RoboDK station: M301_01.rdk

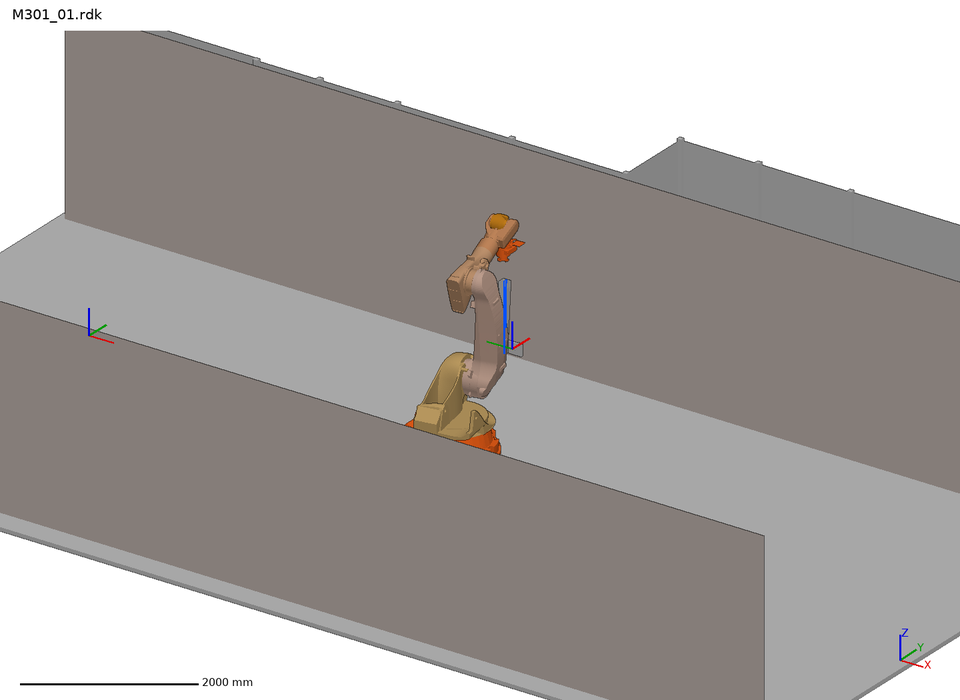
[picture v0: the station drawn from its stored meshes, robots at their saved joint values, targets as dots, program paths as lines]
Station CTTLab. Poses are relative to the parent item; angles as X-Y-Z fixed-axis rotations.
  - object PLANCHER at (0, 0, 0) mm, size 14365 x 8134 x 50 mm, geometry from PLANCHER.STL
  - object BARRIERE_POTEAU at (0, 0, 0) mm, size 13974 x 1274 x 2640 mm, geometry from BARRIERE_POTEAU.STL
  - object BARRIERE_GRILLAGE at (0, 0, 0) mm, size 13811.6 x 1129 x 2475 mm, geometry from BARRIERE_GRILLAGE.STL
  - object BARRIERE_IMMATERIELLE at (0, 0, 0) mm, size 14165 x 6570 x 2640 mm, geometry from BARRIERE_IMMATERIELLE.STL
  - frame World Base at (0, 0, 2.5) mm
    - robot Linear Rail: 1 axes
        modified DH rows (alpha deg, a mm, theta deg, d mm): 0, 0, 0, 0 linear
        base shift (0, 0, 0) mm, rotated rx 0 ry 90 rz 0 deg
        joint limits [0] to [7000]; home [0]; saved at [5000]
      - robot KUKA KR 100 HA: 6 axes
          modified DH rows (alpha deg, a mm, theta deg, d mm): 0, 0, 0, 750; -90, 350, 0, 0; 0, 1250, -90, 0; -90, -45, 0, 1000; 90, 0, 0, 0; -90, 0, 180, 210
          joint limits [-185, -120, -119, -350, -125, -350] to [185, 70, 155, 350, 125, 350]; home [0, -90, 90, 0, 0, 0]; saved at [-97.744, -95.279, 76.837, 0, 108.443, -187.744]
        - tool Tool 1, TCP at (13, 8, 496) mm, size 290.8 x 416.4 x 279.8 mm, geometry from OUTIL.STL
          - object M301_01 at (0, 0, 0) mm, size 101.6 x 101.6 x 914.4 mm, geometry from M301_01.stl
  - frame Camera base at (4846.59, 1350.74, 651.46) mm, rotated rx 0 ry 0 rz 90 deg
    - object Camera at (0, 0, 0) mm, rotated rx 90 ry 0 rz 90 deg, size 220 x 170 x 50 mm, geometry from Camera.stl
    - target Approach target (Cartesian target) at (-112.7, 0, 313.4) mm, rotated rx -180 ry 0 rz -90 deg; joints [-97.607, -91.723, 108.46, 0, 73.263, 82.393, 5000] of KUKA KR 100 HA
    - target Target 0 (Cartesian target) at (-112.7, 0, 881.94) mm, rotated rx -180 ry 0 rz -90 deg; joints [-97.607, -92.983, 76.617, 0, 106.366, 82.393, 5000] of KUKA KR 100 HA
    - target Target 1 (Cartesian target) at (-124.95, 0, 850.56) mm, rotated rx -180 ry 0 rz -90 deg; joints [-97.744, -94.315, 79.678, 0.115, 103.822, 82.256, 5000] of KUKA KR 100 HA
    - target Target 2 (Cartesian target) at (-139.47, 0, 817.45) mm, rotated rx -177.14 ry 0 rz -90 deg; joints [-97.914, -95.806, 82.96, 0.254, 101.05, 82.172, 5000] of KUKA KR 100 HA
    - target Target 3 (Cartesian target) at (-154.54, 0, 817.31) mm, rotated rx -177.14 ry 0 rz -90 deg; joints [-98.102, -97.065, 84.055, 0.41, 100.176, 81.98, 5000] of KUKA KR 100 HA
    - target Target 4 (Cartesian target) at (-154.54, 0, 785.81) mm, rotated rx -177.14 ry 0 rz -90 deg; joints [-98.102, -97.304, 86.085, 0.408, 98.386, 81.967, 5000] of KUKA KR 100 HA
    - target Target 5 (Cartesian target) at (-154.54, 0, 785.81) mm, rotated rx -177.14 ry 0 rz -90 deg; joints [-98.102, -97.304, 86.085, 0.408, 98.386, 81.967, 5000] of KUKA KR 100 HA
    - target Target 6 (Cartesian target) at (-154.54, 0, 754.31) mm, rotated rx -177.14 ry 0 rz -90 deg; joints [-98.102, -97.499, 88.067, 0.406, 96.598, 81.955, 5000] of KUKA KR 100 HA
    - target Target 7 (Cartesian target) at (-154.54, 0, 754.31) mm, rotated rx -177.14 ry 0 rz -90 deg; joints [-98.102, -97.499, 88.067, 0.406, 96.598, 81.955, 5000] of KUKA KR 100 HA
    - target Target 8 (Cartesian target) at (-154.54, 0, 722.81) mm, rotated rx -177.14 ry 0 rz -90 deg; joints [-98.102, -97.649, 90.006, 0.405, 94.81, 81.942, 5000] of KUKA KR 100 HA
    - target Target 9 (Cartesian target) at (-154.54, 0, 722.81) mm, rotated rx -177.14 ry 0 rz -90 deg; joints [-98.102, -97.649, 90.006, 0.405, 94.81, 81.942, 5000] of KUKA KR 100 HA
    - target Target 10 (Cartesian target) at (-154.54, 0, 691.3) mm, rotated rx -177.14 ry 0 rz -90 deg; joints [-98.102, -97.754, 91.901, 0.404, 93.019, 81.929, 5000] of KUKA KR 100 HA
    - target Target 11 (Cartesian target) at (-154.54, 0, 691.3) mm, rotated rx -177.14 ry 0 rz -90 deg; joints [-98.102, -97.754, 91.901, 0.404, 93.019, 81.929, 5000] of KUKA KR 100 HA
    - target Target 12 (Cartesian target) at (-154.54, 0, 659.8) mm, rotated rx -177.14 ry 0 rz -90 deg; joints [-98.102, -97.815, 93.756, 0.403, 91.225, 81.917, 5000] of KUKA KR 100 HA
    - target Target 13 (Cartesian target) at (-154.54, 0, 659.8) mm, rotated rx -177.14 ry 0 rz -90 deg; joints [-98.102, -97.815, 93.756, 0.403, 91.225, 81.917, 5000] of KUKA KR 100 HA
    - target Target 14 (Cartesian target) at (-154.54, 0, 628.3) mm, rotated rx -177.14 ry 0 rz -90 deg; joints [-98.102, -97.829, 95.571, 0.403, 89.424, 81.904, 5000] of KUKA KR 100 HA
    - target Target 15 (Cartesian target) at (-154.54, 0, 628.3) mm, rotated rx -177.14 ry 0 rz -90 deg; joints [-98.102, -97.829, 95.571, 0.403, 89.424, 81.904, 5000] of KUKA KR 100 HA
    - target Target 16 (Cartesian target) at (-154.54, 0, 596.8) mm, rotated rx -177.14 ry 0 rz -90 deg; joints [-98.102, -97.798, 97.349, 0.404, 87.615, 81.891, 5000] of KUKA KR 100 HA
    - target Target 17 (Cartesian target) at (-154.54, 0, 596.8) mm, rotated rx -177.14 ry 0 rz -90 deg; joints [-98.102, -97.798, 97.349, 0.404, 87.615, 81.891, 5000] of KUKA KR 100 HA
    - target Target 18 (Cartesian target) at (-154.54, 0, 565.3) mm, rotated rx -177.14 ry 0 rz -90 deg; joints [-98.102, -97.72, 99.09, 0.404, 85.797, 81.878, 5000] of KUKA KR 100 HA
    - target Target 19 (Cartesian target) at (-154.54, 0, 565.3) mm, rotated rx -177.14 ry 0 rz -90 deg; joints [-98.102, -97.72, 99.09, 0.404, 85.797, 81.878, 5000] of KUKA KR 100 HA
    - target Target 20 (Cartesian target) at (-154.54, 0, 533.8) mm, rotated rx -177.14 ry 0 rz -90 deg; joints [-98.102, -97.595, 100.795, 0.405, 83.966, 81.865, 5000] of KUKA KR 100 HA
    - target Target 21 (Cartesian target) at (-154.54, 0, 533.8) mm, rotated rx -177.14 ry 0 rz -90 deg; joints [-98.102, -97.595, 100.795, 0.405, 83.966, 81.865, 5000] of KUKA KR 100 HA
    - target Target 22 (Cartesian target) at (-154.54, 0, 502.3) mm, rotated rx -177.14 ry 0 rz -90 deg; joints [-98.102, -97.421, 102.465, 0.407, 82.122, 81.852, 5000] of KUKA KR 100 HA
    - target Target 23 (Cartesian target) at (-154.54, 0, 502.3) mm, rotated rx -177.14 ry 0 rz -90 deg; joints [-98.102, -97.421, 102.465, 0.407, 82.122, 81.852, 5000] of KUKA KR 100 HA
    - target Target 24 (Cartesian target) at (-154.54, 0, 470.79) mm, rotated rx -177.14 ry 0 rz -90 deg; joints [-98.102, -97.198, 104.102, 0.409, 80.263, 81.839, 5000] of KUKA KR 100 HA
    - target Target 25 (Cartesian target) at (-154.54, 0, 470.79) mm, rotated rx -177.14 ry 0 rz -90 deg; joints [-98.102, -97.198, 104.102, 0.409, 80.263, 81.839, 5000] of KUKA KR 100 HA
    - target Target 26 (Cartesian target) at (-154.54, 0, 439.29) mm, rotated rx -177.14 ry 0 rz -90 deg; joints [-98.102, -96.924, 105.704, 0.412, 78.387, 81.825, 5000] of KUKA KR 100 HA
    - target Target 27 (Cartesian target) at (-154.54, 0, 439.29) mm, rotated rx -177.14 ry 0 rz -90 deg; joints [-98.102, -96.924, 105.704, 0.412, 78.387, 81.825, 5000] of KUKA KR 100 HA
    - target Target 28 (Cartesian target) at (-154.54, 0, 407.79) mm, rotated rx -177.14 ry 0 rz -90 deg; joints [-98.102, -96.599, 107.273, 0.415, 76.492, 81.811, 5000] of KUKA KR 100 HA
    - target Target 29 (Cartesian target) at (-154.54, 0, 407.79) mm, rotated rx -177.14 ry 0 rz -90 deg; joints [-98.102, -96.599, 107.273, 0.415, 76.492, 81.811, 5000] of KUKA KR 100 HA
    - target Target 30 (Cartesian target) at (-154.54, 0, 376.29) mm, rotated rx -177.14 ry 0 rz -90 deg; joints [-98.102, -96.22, 108.809, 0.418, 74.578, 81.797, 5000] of KUKA KR 100 HA
    - target Target 31 (Cartesian target) at (-154.54, 0, 376.29) mm, rotated rx -177.14 ry 0 rz -90 deg; joints [-98.102, -96.22, 108.809, 0.418, 74.578, 81.797, 5000] of KUKA KR 100 HA
    - target Target 32 (Cartesian target) at (-154.54, 0, 344.79) mm, rotated rx -177.14 ry 0 rz -90 deg; joints [-98.102, -95.787, 110.312, 0.422, 72.642, 81.782, 5000] of KUKA KR 100 HA
    - target Target 33 (Cartesian target) at (-154.54, 0, 344.79) mm, rotated rx -177.14 ry 0 rz -90 deg; joints [-98.102, -95.787, 110.312, 0.422, 72.642, 81.782, 5000] of KUKA KR 100 HA
    - target Target 34 (Cartesian target) at (-154.54, 0, 313.29) mm, rotated rx -177.14 ry 0 rz -90 deg; joints [-98.102, -95.298, 111.781, 0.427, 70.683, 81.767, 5000] of KUKA KR 100 HA
    - target Target 35 (Cartesian target) at (-154.54, 0, 313.29) mm, rotated rx -177.14 ry 0 rz -90 deg; joints [-98.102, -95.298, 111.781, 0.427, 70.683, 81.767, 5000] of KUKA KR 100 HA
    - target Target 36 (Cartesian target) at (-154.54, 0, 281.79) mm, rotated rx -177.14 ry 0 rz -90 deg; joints [-98.102, -94.751, 113.218, 0.433, 68.7, 81.751, 5000] of KUKA KR 100 HA
    - target Target 37 (Cartesian target) at (-154.54, 0, 281.79) mm, rotated rx -177.14 ry 0 rz -90 deg; joints [-98.102, -94.751, 113.218, 0.433, 68.7, 81.751, 5000] of KUKA KR 100 HA
    - target Target 38 (Cartesian target) at (-154.54, 0, 250.29) mm, rotated rx -177.14 ry 0 rz -90 deg; joints [-98.102, -94.146, 114.621, 0.439, 66.691, 81.734, 5000] of KUKA KR 100 HA
    - target Target 39 (Cartesian target) at (-154.54, 0, 218.78) mm, rotated rx -177.14 ry 0 rz -90 deg; joints [-98.102, -93.479, 115.99, 0.446, 64.656, 81.717, 5000] of KUKA KR 100 HA
    - target Target 40 (Cartesian target) at (-154.54, 0, 218.78) mm, rotated rx -177.14 ry 0 rz -90 deg; joints [-98.102, -93.479, 115.99, 0.446, 64.656, 81.717, 5000] of KUKA KR 100 HA
    - target Target 41 (Cartesian target) at (-154.54, 0, 187.28) mm, rotated rx -177.14 ry 0 rz -90 deg; joints [-98.102, -92.751, 117.325, 0.454, 62.593, 81.699, 5000] of KUKA KR 100 HA
    - target Target 42 (Cartesian target) at (-154.54, 0, 187.28) mm, rotated rx -177.14 ry 0 rz -90 deg; joints [-98.102, -92.751, 117.325, 0.454, 62.593, 81.699, 5000] of KUKA KR 100 HA
    - target Target 43 (Cartesian target) at (-154.54, 0, 155.78) mm, rotated rx -177.14 ry 0 rz -90 deg; joints [81.898, -118.157, -84.385, 0.446, -64.624, -98.283, 5000] of KUKA KR 100 HA
    - target Target 44 (Cartesian target) at (-154.54, 0, 155.78) mm, rotated rx -177.14 ry 0 rz -90 deg; joints [81.898, -118.157, -84.385, 0.446, -64.624, -98.283, 5000] of KUKA KR 100 HA
    - target Target 45 (Cartesian target) at (-154.54, 0, 124.28) mm, rotated rx -177.14 ry 0 rz -90 deg; joints [81.898, -118.674, -85.469, 0.452, -63.024, -98.297, 5000] of KUKA KR 100 HA
    - target Target 46 (Cartesian target) at (-154.54, 0, 124.28) mm, rotated rx -177.14 ry 0 rz -90 deg; joints [81.898, -118.674, -85.469, 0.452, -63.024, -98.297, 5000] of KUKA KR 100 HA
    - target Target 47 (Cartesian target) at (-154.54, 0, 92.78) mm, rotated rx -177.14 ry 0 rz -90 deg; joints [81.898, -119.227, -86.504, 0.459, -61.436, -98.312, 5000] of KUKA KR 100 HA
    - target Target 48 (Cartesian target) at (-152.66, 0, 92.8) mm, rotated rx -177.14 ry 0 rz -90 deg; joints [82.007, -119.904, -85.364, 0.266, -63.062, -98.187, 5000] of KUKA KR 100 HA
    - target Target 49 (Cartesian target) at (-151.82, 0, 63.93) mm, rotated rx -180 ry 0 rz -90 deg; joints [-97.923, -88.095, 120.951, 0.152, 56.229, 82.077, 5000] of KUKA KR 100 HA
    - target Target 50 (Cartesian target) at (-150.8, 0, 32.46) mm, rotated rx -180 ry 0 rz -90 deg; joints [-97.844, -86.52, 121.508, 0, 55.012, 82.156, 5000] of KUKA KR 100 HA
    - target Target 51 (Cartesian target) at (-150.8, 0, 1) mm, rotated rx -180 ry 0 rz -90 deg; joints [-97.844, -85.425, 122.596, 0, 52.829, 82.156, 5000] of KUKA KR 100 HA
    - target Target 52 (Cartesian target) at (-150.8, 0, 1) mm, rotated rx -180 ry 0 rz 180 deg; joints [-96.836, -85.327, 122.485, 0, 52.842, -6.836, 5000] of KUKA KR 100 HA
    - target Target 53 (Cartesian target) at (-150.8, 0, 32.46) mm, rotated rx -180 ry 0 rz 180 deg; joints [-96.836, -86.42, 121.398, 0, 55.022, -6.836, 5000] of KUKA KR 100 HA
    - target Target 54 (Cartesian target) at (-150.8, 0, 63.92) mm, rotated rx -180 ry 0 rz 180 deg; joints [-96.836, -87.447, 120.271, 0, 57.176, -6.836, 5000] of KUKA KR 100 HA
    - target Target 55 (Cartesian target) at (-150.8, 0, 95.39) mm, rotated rx -180 ry 0 rz 180 deg; joints [-96.836, -88.409, 119.105, 0, 59.305, -6.836, 5000] of KUKA KR 100 HA
    - target Target 56 (Cartesian target) at (-150.8, 0, 126.85) mm, rotated rx -180 ry 0 rz 180 deg; joints [-96.836, -89.307, 117.9, 0, 61.407, -6.836, 5000] of KUKA KR 100 HA
    - target Target 57 (Cartesian target) at (-150.8, 0, 158.31) mm, rotated rx -180 ry 0 rz 180 deg; joints [-96.836, -90.142, 116.658, 0, 63.483, -6.836, 5000] of KUKA KR 100 HA
    - target Target 58 (Cartesian target) at (-150.8, 0, 189.77) mm, rotated rx -180 ry 0 rz 180 deg; joints [-96.836, -90.915, 115.38, 0, 65.535, -6.836, 5000] of KUKA KR 100 HA
    - target Target 59 (Cartesian target) at (-150.8, 0, 221.23) mm, rotated rx -180 ry 0 rz 180 deg; joints [-96.836, -91.627, 114.066, 0, 67.561, -6.836, 5000] of KUKA KR 100 HA
    - target Target 60 (Cartesian target) at (-150.8, 0, 252.7) mm, rotated rx -180 ry 0 rz 180 deg; joints [-96.836, -92.28, 112.717, 0, 69.563, -6.836, 5000] of KUKA KR 100 HA
    - target Target 61 (Cartesian target) at (-150.8, 0, 284.16) mm, rotated rx -180 ry 0 rz 180 deg; joints [-96.836, -92.874, 111.333, 0, 71.541, -6.836, 5000] of KUKA KR 100 HA
    - target Target 62 (Cartesian target) at (-150.8, 0, 315.62) mm, rotated rx -180 ry 0 rz 180 deg; joints [-96.836, -93.412, 109.915, 0, 73.498, -6.836, 5000] of KUKA KR 100 HA
    - target Target 63 (Cartesian target) at (-150.8, 0, 347.08) mm, rotated rx -180 ry 0 rz 180 deg; joints [-96.836, -93.895, 108.462, 0, 75.433, -6.836, 5000] of KUKA KR 100 HA
    - target Target 64 (Cartesian target) at (-150.8, 0, 378.54) mm, rotated rx -180 ry 0 rz 180 deg; joints [-96.836, -94.324, 106.976, 0, 77.348, -6.836, 5000] of KUKA KR 100 HA
    - target Target 65 (Cartesian target) at (-150.8, 0, 410.01) mm, rotated rx -180 ry 0 rz 180 deg; joints [-96.836, -94.699, 105.455, 0, 79.245, -6.836, 5000] of KUKA KR 100 HA
    - target Target 66 (Cartesian target) at (-150.8, 0, 441.47) mm, rotated rx -180 ry 0 rz 180 deg; joints [-96.836, -95.024, 103.9, 0, 81.124, -6.836, 5000] of KUKA KR 100 HA
    - target Target 67 (Cartesian target) at (-150.8, 0, 472.93) mm, rotated rx -180 ry 0 rz 180 deg; joints [-96.836, -95.297, 102.311, 0, 82.986, -6.836, 5000] of KUKA KR 100 HA
    - target Target 68 (Cartesian target) at (-150.8, 0, 504.39) mm, rotated rx -180 ry 0 rz 180 deg; joints [-96.836, -95.521, 100.686, 0, 84.835, -6.836, 5000] of KUKA KR 100 HA
    - target Target 69 (Cartesian target) at (-150.8, 0, 535.86) mm, rotated rx -180 ry 0 rz 180 deg; joints [-96.836, -95.697, 99.026, 0, 86.67, -6.836, 5000] of KUKA KR 100 HA
    - target Target 70 (Cartesian target) at (-150.8, 0, 567.32) mm, rotated rx -180 ry 0 rz 180 deg; joints [-96.836, -95.824, 97.33, 0, 88.494, -6.836, 5000] of KUKA KR 100 HA
    - target Target 71 (Cartesian target) at (-150.8, 0, 598.78) mm, rotated rx -180 ry 0 rz 180 deg; joints [-96.836, -95.905, 95.597, 0, 90.308, -6.836, 5000] of KUKA KR 100 HA
    - target Target 72 (Cartesian target) at (-150.8, 0, 630.24) mm, rotated rx -180 ry 0 rz 180 deg; joints [-96.836, -95.94, 93.826, 0, 92.114, -6.836, 5000] of KUKA KR 100 HA
    - target Target 73 (Cartesian target) at (-150.8, 0, 661.7) mm, rotated rx -180 ry 0 rz 180 deg; joints [-96.836, -95.929, 92.015, 0, 93.913, -6.836, 5000] of KUKA KR 100 HA
    - target Target 74 (Cartesian target) at (-150.8, 0, 693.17) mm, rotated rx -180 ry 0 rz 180 deg; joints [-96.836, -95.872, 90.164, 0, 95.708, -6.836, 5000] of KUKA KR 100 HA
    - target Target 75 (Cartesian target) at (-150.8, 0, 724.63) mm, rotated rx -180 ry 0 rz 180 deg; joints [-96.836, -95.771, 88.27, 0, 97.501, -6.836, 5000] of KUKA KR 100 HA
    - target Target 76 (Cartesian target) at (-150.8, 0, 756.09) mm, rotated rx -180 ry 0 rz 180 deg; joints [-96.836, -95.625, 86.332, 0, 99.293, -6.836, 5000] of KUKA KR 100 HA
    - target Target 77 (Cartesian target) at (-150.8, 0, 787.55) mm, rotated rx -180 ry 0 rz 180 deg; joints [-96.836, -95.434, 84.347, 0, 101.087, -6.836, 5000] of KUKA KR 100 HA
    - target Target 78 (Cartesian target) at (-150.8, 0, 819.01) mm, rotated rx -180 ry 0 rz 180 deg; joints [-96.836, -95.197, 82.313, 0, 102.884, -6.836, 5000] of KUKA KR 100 HA
    - target Target 79 (Cartesian target) at (-150.8, 0, 850.48) mm, rotated rx -180 ry 0 rz 180 deg; joints [-96.836, -94.915, 80.227, 0, 104.689, -6.836, 5000] of KUKA KR 100 HA
    - target Target 80 (Cartesian target) at (-150.8, 0, 881.94) mm, rotated rx -180 ry 0 rz 180 deg; joints [-96.836, -94.587, 78.085, 0, 106.502, -6.836, 5000] of KUKA KR 100 HA
    - target Target 81 (Cartesian target) at (-150.8, 0, 913.4) mm, rotated rx -180 ry 0 rz 180 deg; joints [-96.836, -94.212, 75.884, 0, 108.328, -6.836, 5000] of KUKA KR 100 HA
    - target Target 82 (Cartesian target) at (-112.7, 0, 913.4) mm, rotated rx -180 ry 0 rz 90 deg; joints [-96.512, -93.472, 75.208, 0, 108.264, -96.512, 5000] of KUKA KR 100 HA
    - target Target 83 (Cartesian target) at (-112.7, 0, 881.94) mm, rotated rx -180 ry 0 rz 90 deg; joints [-96.512, -93.847, 77.415, 0, 106.432, -96.512, 5000] of KUKA KR 100 HA
    - target Target 84 (Cartesian target) at (-124.95, 0, 850.56) mm, rotated rx -180 ry 0 rz 90 deg; joints [-96.632, -95.179, 80.451, 0.098, 103.911, -96.632, 5000] of KUKA KR 100 HA
    - target Target 85 (Cartesian target) at (-139.47, 0, 817.45) mm, rotated rx 177.14 ry 0 rz 90 deg; joints [-96.78, -96.68, 83.76, 0.217, 101.119, -96.705, 5000] of KUKA KR 100 HA
    - target Target 86 (Cartesian target) at (-154.54, 0, 817.31) mm, rotated rx 177.14 ry 0 rz 90 deg; joints [-96.943, -97.94, 84.831, 0.352, 100.267, -96.872, 5000] of KUKA KR 100 HA
    - target Target 87 (Cartesian target) at (-154.54, 0, 785.81) mm, rotated rx 177.14 ry 0 rz 90 deg; joints [-96.943, -98.182, 86.859, 0.35, 98.481, -96.883, 5000] of KUKA KR 100 HA
    - target Target 88 (Cartesian target) at (-154.54, 0, 785.81) mm, rotated rx 177.14 ry 0 rz 90 deg; joints [-96.943, -98.182, 86.859, 0.35, 98.481, -96.883, 5000] of KUKA KR 100 HA
    - target Target 89 (Cartesian target) at (-154.54, 0, 754.31) mm, rotated rx 177.14 ry 0 rz 90 deg; joints [-96.943, -98.38, 88.841, 0.348, 96.697, -96.894, 5000] of KUKA KR 100 HA
    - target Target 90 (Cartesian target) at (-154.54, 0, 754.31) mm, rotated rx 177.14 ry 0 rz 90 deg; joints [-96.943, -98.38, 88.841, 0.348, 96.697, -96.894, 5000] of KUKA KR 100 HA
    - target Target 91 (Cartesian target) at (-154.54, 0, 722.81) mm, rotated rx 177.14 ry 0 rz 90 deg; joints [-96.943, -98.532, 90.779, 0.347, 94.912, -96.905, 5000] of KUKA KR 100 HA
    - target Target 92 (Cartesian target) at (-154.54, 0, 722.81) mm, rotated rx 177.14 ry 0 rz 90 deg; joints [-96.943, -98.532, 90.779, 0.347, 94.912, -96.905, 5000] of KUKA KR 100 HA
    - target Target 93 (Cartesian target) at (-154.54, 0, 691.3) mm, rotated rx 177.14 ry 0 rz 90 deg; joints [-96.943, -98.64, 92.675, 0.346, 93.124, -96.916, 5000] of KUKA KR 100 HA
    - target Target 94 (Cartesian target) at (-154.54, 0, 691.3) mm, rotated rx 177.14 ry 0 rz 90 deg; joints [-96.943, -98.64, 92.675, 0.346, 93.124, -96.916, 5000] of KUKA KR 100 HA
    - target Target 95 (Cartesian target) at (-154.54, 0, 659.8) mm, rotated rx 177.14 ry 0 rz 90 deg; joints [-96.943, -98.704, 94.531, 0.346, 91.331, -96.927, 5000] of KUKA KR 100 HA
    - target Target 96 (Cartesian target) at (-154.54, 0, 659.8) mm, rotated rx 177.14 ry 0 rz 90 deg; joints [-96.943, -98.704, 94.531, 0.346, 91.331, -96.927, 5000] of KUKA KR 100 HA
    - target Target 97 (Cartesian target) at (-154.54, 0, 628.3) mm, rotated rx 177.14 ry 0 rz 90 deg; joints [-96.943, -98.721, 96.349, 0.346, 89.531, -96.938, 5000] of KUKA KR 100 HA
    - target Target 98 (Cartesian target) at (-154.54, 0, 628.3) mm, rotated rx 177.14 ry 0 rz 90 deg; joints [-96.943, -98.721, 96.349, 0.346, 89.531, -96.938, 5000] of KUKA KR 100 HA
    - target Target 99 (Cartesian target) at (-154.54, 0, 596.8) mm, rotated rx 177.14 ry 0 rz 90 deg; joints [-96.943, -98.693, 98.129, 0.346, 87.722, -96.948, 5000] of KUKA KR 100 HA
    - target Target 100 (Cartesian target) at (-154.54, 0, 596.8) mm, rotated rx 177.14 ry 0 rz 90 deg; joints [-96.943, -98.693, 98.129, 0.346, 87.722, -96.948, 5000] of KUKA KR 100 HA
    - target Target 101 (Cartesian target) at (-154.54, 0, 565.3) mm, rotated rx 177.14 ry 0 rz 90 deg; joints [-96.943, -98.618, 99.874, 0.347, 85.903, -96.959, 5000] of KUKA KR 100 HA
    - target Target 102 (Cartesian target) at (-154.54, 0, 565.3) mm, rotated rx 177.14 ry 0 rz 90 deg; joints [-96.943, -98.618, 99.874, 0.347, 85.903, -96.959, 5000] of KUKA KR 100 HA
    - target Target 103 (Cartesian target) at (-154.54, 0, 533.8) mm, rotated rx 177.14 ry 0 rz 90 deg; joints [-96.943, -98.495, 101.583, 0.348, 84.071, -96.971, 5000] of KUKA KR 100 HA
    - target Target 104 (Cartesian target) at (-154.54, 0, 533.8) mm, rotated rx 177.14 ry 0 rz 90 deg; joints [-96.943, -98.495, 101.583, 0.348, 84.071, -96.971, 5000] of KUKA KR 100 HA
    - target Target 105 (Cartesian target) at (-154.54, 0, 502.3) mm, rotated rx 177.14 ry 0 rz 90 deg; joints [-96.943, -98.324, 103.258, 0.349, 82.224, -96.982, 5000] of KUKA KR 100 HA
    - target Target 106 (Cartesian target) at (-154.54, 0, 502.3) mm, rotated rx 177.14 ry 0 rz 90 deg; joints [-96.943, -98.324, 103.258, 0.349, 82.224, -96.982, 5000] of KUKA KR 100 HA
    - target Target 107 (Cartesian target) at (-154.54, 0, 470.79) mm, rotated rx 177.14 ry 0 rz 90 deg; joints [-96.943, -98.102, 104.9, 0.351, 80.361, -96.993, 5000] of KUKA KR 100 HA
    - target Target 108 (Cartesian target) at (-154.54, 0, 470.79) mm, rotated rx 177.14 ry 0 rz 90 deg; joints [-96.943, -98.102, 104.9, 0.351, 80.361, -96.993, 5000] of KUKA KR 100 HA
    - target Target 109 (Cartesian target) at (-154.54, 0, 439.29) mm, rotated rx 177.14 ry 0 rz 90 deg; joints [-96.943, -97.83, 106.508, 0.353, 78.481, -97.005, 5000] of KUKA KR 100 HA
    - target Target 110 (Cartesian target) at (-154.54, 0, 439.29) mm, rotated rx 177.14 ry 0 rz 90 deg; joints [-96.943, -97.83, 106.508, 0.353, 78.481, -97.005, 5000] of KUKA KR 100 HA
    - target Target 111 (Cartesian target) at (-154.54, 0, 407.79) mm, rotated rx 177.14 ry 0 rz 90 deg; joints [-96.943, -97.505, 108.084, 0.356, 76.58, -97.017, 5000] of KUKA KR 100 HA
    - target Target 112 (Cartesian target) at (-154.54, 0, 407.79) mm, rotated rx 177.14 ry 0 rz 90 deg; joints [-96.943, -97.505, 108.084, 0.356, 76.58, -97.017, 5000] of KUKA KR 100 HA
    - target Target 113 (Cartesian target) at (-154.54, 0, 376.29) mm, rotated rx 177.14 ry 0 rz 90 deg; joints [-96.943, -97.127, 109.627, 0.359, 74.659, -97.03, 5000] of KUKA KR 100 HA
    - target Target 114 (Cartesian target) at (-154.54, 0, 376.29) mm, rotated rx 177.14 ry 0 rz 90 deg; joints [-96.943, -97.127, 109.627, 0.359, 74.659, -97.03, 5000] of KUKA KR 100 HA
    - target Target 115 (Cartesian target) at (-154.54, 0, 344.79) mm, rotated rx 177.14 ry 0 rz 90 deg; joints [-96.943, -96.694, 111.137, 0.362, 72.715, -97.042, 5000] of KUKA KR 100 HA
    - target Target 116 (Cartesian target) at (-154.54, 0, 344.79) mm, rotated rx 177.14 ry 0 rz 90 deg; joints [-96.943, -96.694, 111.137, 0.362, 72.715, -97.042, 5000] of KUKA KR 100 HA
    - target Target 117 (Cartesian target) at (-154.54, 0, 313.29) mm, rotated rx 177.14 ry 0 rz 90 deg; joints [-96.943, -96.203, 112.615, 0.366, 70.747, -97.056, 5000] of KUKA KR 100 HA
    - target Target 118 (Cartesian target) at (-154.54, 0, 313.29) mm, rotated rx 177.14 ry 0 rz 90 deg; joints [-96.943, -96.203, 112.615, 0.366, 70.747, -97.056, 5000] of KUKA KR 100 HA
    - target Target 119 (Cartesian target) at (-154.54, 0, 281.79) mm, rotated rx 177.14 ry 0 rz 90 deg; joints [-96.943, -95.655, 114.061, 0.371, 68.753, -97.069, 5000] of KUKA KR 100 HA
    - target Target 120 (Cartesian target) at (-154.54, 0, 281.79) mm, rotated rx 177.14 ry 0 rz 90 deg; joints [-96.943, -95.655, 114.061, 0.371, 68.753, -97.069, 5000] of KUKA KR 100 HA
    - target Target 121 (Cartesian target) at (-154.54, 0, 250.29) mm, rotated rx 177.14 ry 0 rz 90 deg; joints [-96.943, -95.046, 115.473, 0.377, 66.732, -97.083, 5000] of KUKA KR 100 HA
    - target Target 122 (Cartesian target) at (-154.54, 0, 218.78) mm, rotated rx 177.14 ry 0 rz 90 deg; joints [83.057, -116.391, -83.461, 0.375, -67.307, 82.921, 5000] of KUKA KR 100 HA
    - target Target 123 (Cartesian target) at (-154.54, 0, 218.78) mm, rotated rx 177.14 ry 0 rz 90 deg; joints [83.057, -116.391, -83.461, 0.375, -67.307, 82.921, 5000] of KUKA KR 100 HA
    - target Target 124 (Cartesian target) at (-154.54, 0, 187.28) mm, rotated rx 177.14 ry 0 rz 90 deg; joints [83.057, -116.844, -84.638, 0.38, -65.677, 82.909, 5000] of KUKA KR 100 HA
    - target Target 125 (Cartesian target) at (-154.54, 0, 187.28) mm, rotated rx 177.14 ry 0 rz 90 deg; joints [83.057, -116.844, -84.638, 0.38, -65.677, 82.909, 5000] of KUKA KR 100 HA
    - target Target 126 (Cartesian target) at (-154.54, 0, 155.78) mm, rotated rx 177.14 ry 0 rz 90 deg; joints [83.057, -117.335, -85.765, 0.385, -64.059, 82.897, 5000] of KUKA KR 100 HA
    - target Target 127 (Cartesian target) at (-154.54, 0, 155.78) mm, rotated rx 177.14 ry 0 rz 90 deg; joints [83.057, -117.335, -85.765, 0.385, -64.059, 82.897, 5000] of KUKA KR 100 HA
    - target Target 128 (Cartesian target) at (-154.54, 0, 124.28) mm, rotated rx 177.14 ry 0 rz 90 deg; joints [83.057, -117.864, -86.845, 0.39, -62.451, 82.885, 5000] of KUKA KR 100 HA
    - target Target 129 (Cartesian target) at (-154.54, 0, 124.28) mm, rotated rx 177.14 ry 0 rz 90 deg; joints [83.057, -117.864, -86.845, 0.39, -62.451, 82.885, 5000] of KUKA KR 100 HA
    - target Target 130 (Cartesian target) at (-154.54, 0, 92.78) mm, rotated rx 177.14 ry 0 rz 90 deg; joints [83.057, -118.428, -87.876, 0.396, -60.855, 82.872, 5000] of KUKA KR 100 HA
    - target Target 131 (Cartesian target) at (-152.66, 0, 92.8) mm, rotated rx 177.14 ry 0 rz 90 deg; joints [83.152, -119.102, -86.752, 0.229, -62.472, 82.981, 5000] of KUKA KR 100 HA
    - target Target 132 (Cartesian target) at (-151.82, 0, 63.93) mm, rotated rx -180 ry 0 rz 90 deg; joints [-96.788, -88.96, 121.849, 0.13, 56.193, -96.788, 5000] of KUKA KR 100 HA
    - target Target 133 (Cartesian target) at (-150.8, 0, 32.46) mm, rotated rx -180 ry 0 rz 90 deg; joints [-96.718, -87.365, 122.424, 0, 54.941, -96.718, 5000] of KUKA KR 100 HA
    - target Target 134 (Cartesian target) at (-150.8, 0, 1) mm, rotated rx -180 ry 0 rz 90 deg; joints [-96.718, -86.256, 123.525, 0, 52.731, -96.718, 5000] of KUKA KR 100 HA
    - target Target 135 (Cartesian target) at (-150.8, 0, 1) mm, rotated rx -180 ry 0 rz 0 deg; joints [-97.744, -86.357, 123.636, 0, 52.72, 172.256, 5000] of KUKA KR 100 HA
    - target Target 136 (Cartesian target) at (-150.8, 0, 32.46) mm, rotated rx -180 ry 0 rz 0 deg; joints [-97.744, -87.468, 122.534, 0, 54.934, 172.256, 5000] of KUKA KR 100 HA
    - target Target 137 (Cartesian target) at (-150.8, 0, 63.92) mm, rotated rx -180 ry 0 rz 0 deg; joints [-97.744, -88.51, 121.392, 0, 57.119, 172.256, 5000] of KUKA KR 100 HA
    - target Target 138 (Cartesian target) at (-150.8, 0, 95.39) mm, rotated rx -180 ry 0 rz 0 deg; joints [82.256, -119.901, -85.187, 0, -64.912, -7.744, 5000] of KUKA KR 100 HA
    - target Target 139 (Cartesian target) at (-150.8, 0, 126.85) mm, rotated rx -180 ry 0 rz 0 deg; joints [82.256, -119.362, -84.146, 0, -66.492, -7.744, 5000] of KUKA KR 100 HA
    - target Target 140 (Cartesian target) at (-150.8, 0, 158.31) mm, rotated rx -180 ry 0 rz 0 deg; joints [82.256, -118.86, -83.056, 0, -68.085, -7.744, 5000] of KUKA KR 100 HA
    - target Target 141 (Cartesian target) at (-150.8, 0, 189.77) mm, rotated rx -180 ry 0 rz 0 deg; joints [82.256, -118.394, -81.916, 0, -69.691, -7.744, 5000] of KUKA KR 100 HA
    - target Target 142 (Cartesian target) at (-150.8, 0, 221.23) mm, rotated rx -180 ry 0 rz 0 deg; joints [82.256, -117.966, -80.725, 0, -71.309, -7.744, 5000] of KUKA KR 100 HA
    - target Target 143 (Cartesian target) at (-150.8, 0, 252.7) mm, rotated rx -180 ry 0 rz 0 deg; joints [82.256, -117.576, -79.483, 0, -72.941, -7.744, 5000] of KUKA KR 100 HA
    - target Target 144 (Cartesian target) at (-150.8, 0, 284.16) mm, rotated rx -180 ry 0 rz 0 deg; joints [82.256, -117.226, -78.187, 0, -74.587, -7.744, 5000] of KUKA KR 100 HA
    - target Target 145 (Cartesian target) at (-150.8, 0, 315.62) mm, rotated rx -180 ry 0 rz 0 deg; joints [82.256, -116.915, -76.837, 0, -76.248, -7.744, 5000] of KUKA KR 100 HA
    - target Target 146 (Cartesian target) at (-150.8, 0, 347.08) mm, rotated rx -180 ry 0 rz 0 deg; joints [82.256, -116.645, -75.431, 0, -77.924, -7.744, 5000] of KUKA KR 100 HA
    - target Target 147 (Cartesian target) at (-150.8, 0, 378.54) mm, rotated rx -180 ry 0 rz 0 deg; joints [82.256, -116.417, -73.966, 0, -79.617, -7.744, 5000] of KUKA KR 100 HA
    - target Target 148 (Cartesian target) at (-150.8, 0, 410.01) mm, rotated rx -180 ry 0 rz 0 deg; joints [82.256, -116.232, -72.44, 0, -81.328, -7.744, 5000] of KUKA KR 100 HA
    - target Target 149 (Cartesian target) at (-150.8, 0, 441.47) mm, rotated rx -180 ry 0 rz 0 deg; joints [82.256, -116.091, -70.85, 0, -83.059, -7.744, 5000] of KUKA KR 100 HA
    - target Target 150 (Cartesian target) at (-150.8, 0, 472.93) mm, rotated rx -180 ry 0 rz 0 deg; joints [82.256, -115.996, -69.193, 0, -84.811, -7.744, 5000] of KUKA KR 100 HA
    - target Target 151 (Cartesian target) at (-150.8, 0, 504.39) mm, rotated rx -180 ry 0 rz 0 deg; joints [82.256, -115.949, -67.465, 0, -86.586, -7.744, 5000] of KUKA KR 100 HA
    - target Target 152 (Cartesian target) at (-150.8, 0, 535.86) mm, rotated rx -180 ry 0 rz 0 deg; joints [82.256, -115.95, -65.661, 0, -88.388, -7.744, 5000] of KUKA KR 100 HA
    - target Target 153 (Cartesian target) at (-150.8, 0, 567.32) mm, rotated rx -180 ry 0 rz 0 deg; joints [82.256, -116.004, -63.777, 0, -90.219, -7.744, 5000] of KUKA KR 100 HA
    - target Target 154 (Cartesian target) at (-150.8, 0, 598.78) mm, rotated rx -180 ry 0 rz 0 deg; joints [82.256, -116.112, -61.805, 0, -92.083, -7.744, 5000] of KUKA KR 100 HA
    - target Target 155 (Cartesian target) at (-150.8, 0, 630.24) mm, rotated rx -180 ry 0 rz 0 deg; joints [82.256, -116.278, -59.737, 0, -93.985, -7.744, 5000] of KUKA KR 100 HA
    - target Target 156 (Cartesian target) at (-150.8, 0, 661.7) mm, rotated rx -180 ry 0 rz 0 deg; joints [82.256, -116.506, -57.565, 0, -95.929, -7.744, 5000] of KUKA KR 100 HA
    - target Target 157 (Cartesian target) at (-150.8, 0, 693.17) mm, rotated rx -180 ry 0 rz 0 deg; joints [82.256, -116.801, -55.277, 0, -97.922, -7.744, 5000] of KUKA KR 100 HA
    - target Target 158 (Cartesian target) at (-150.8, 0, 724.63) mm, rotated rx -180 ry 0 rz 0 deg; joints [82.256, -117.169, -52.858, 0, -99.973, -7.744, 5000] of KUKA KR 100 HA
    - target Target 159 (Cartesian target) at (-150.8, 0, 756.09) mm, rotated rx -180 ry 0 rz 0 deg; joints [82.256, -117.619, -50.289, 0, -102.092, -7.744, 5000] of KUKA KR 100 HA
    - target Target 160 (Cartesian target) at (-150.8, 0, 787.55) mm, rotated rx -180 ry 0 rz 0 deg; joints [82.256, -118.16, -47.547, 0, -104.292, -7.744, 5000] of KUKA KR 100 HA
    - target Target 161 (Cartesian target) at (-150.8, 0, 819.01) mm, rotated rx -180 ry 0 rz 0 deg; joints [82.256, -118.808, -44.6, 0, -106.592, -7.744, 5000] of KUKA KR 100 HA
    - target Target 162 (Cartesian target) at (-150.8, 0, 850.48) mm, rotated rx -180 ry 0 rz 0 deg; joints [82.256, -119.583, -41.401, 0, -109.017, -7.744, 5000] of KUKA KR 100 HA
    - target Target 163 (Cartesian target) at (-150.8, 0, 881.94) mm, rotated rx -180 ry 0 rz 0 deg; joints [-97.744, -95.657, 79.032, 0, 106.625, 172.256, 5000] of KUKA KR 100 HA
    - target Target 164 (Cartesian target) at (-150.8, 0, 913.4) mm, rotated rx -180 ry 0 rz 0 deg; joints [-97.744, -95.279, 76.837, 0, 108.443, 172.256, 5000] of KUKA KR 100 HA
  - Python program LoadProgram (listed below)
  - Python program UpdateExternalJoints (listed below)
  - program M301_01 Picture Analysis (169 instructions, listed below)
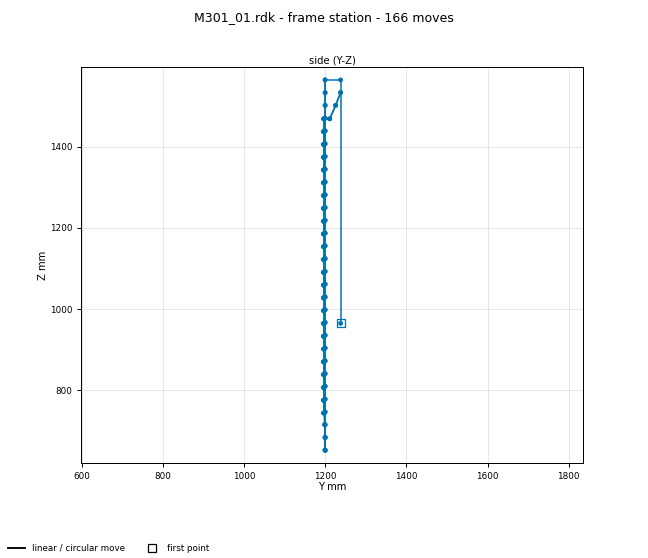
[picture p0: tool path of M301_01.rdk in frame station, 166 of 166 moves have a stored position in this frame; points joined in program order, loops and branches not executed]

--- Python program LoadProgram ---
from robolink import *

RDK = Robolink()

robot = RDK.Item('KUKA KR 100 HA', ITEM_TYPE_ROBOT)
if not robot.Valid():
    raise Exception('No robot selected or available')

world_base = RDK.Item('World Base', ITEM_TYPE_FRAME)
camera_base = RDK.Item('Camera base', ITEM_TYPE_FRAME)
tool = RDK.Item('Tool 1', ITEM_TYPE_TOOL)

RDK.Render(False)


# Specify the reference frame you want to use
program = RDK.AddProgram("{} Picture Analysis".format(name_prog), robot)
program.setPoseFrame(camera_base)
program.setPoseTool(tool)

program.setSpeed(speed, 200, 10000, 800)

target_name = 'Approach target'
pose = Mat(htm[0].tolist())
target = RDK.AddTarget(target_name, camera_base, tool)
target.setAsCartesianTarget()
target.setPose(pose)
program.MoveJ(target)



for i in range(htm.shape[0] - 1):
    target_name = 'Target {}'.format(i)
    pose = Mat(htm[i + 1].tolist())
    target = RDK.AddTarget(target_name, camera_base, tool)
    e1 = 5000
    target.setJoints([0,0,0,0,0,0, e1])
    target.setAsCartesianTarget()
    target.setPose(pose)
    program.MoveL(target)

--- Python program UpdateExternalJoints ---
# Type help("robolink") or help("robodk") for more information
# Press F5 to run the script
# Documentation: https://robodk.com/doc/en/RoboDK-API.html
# Reference:     https://robodk.com/doc/en/PythonAPI/index.html
# Note: It is not required to keep a copy of this file, your python script is saved with the station
from robolink import *    # RoboDK API
from robodk import *      # Robot toolbox
RDK = Robolink()

targets = RDK.ItemList(ITEM_TYPE_TARGET)

RDK.Render(False)
for t in targets:
    # Set the value of the external axis
    e1 = 5000 # in mm
    t.setJoints([0,0,0,0,0,0, e1])

    # Recalculate the joint position based on the new position of the external axis
    # Robot joints are updated but not external axis
    t.setAsCartesianTarget()
    t.Joints()

    jnts = t.Joints()
    print(t.Name() + "-Joints: " + str(jnts.list()))

--- program M301_01 Picture Analysis (robot KUKA KR 100 HA) ---
  Set Ref.: Camera base
  Choisir Outil: Tool 1
  Set speed (50.0 mm/s)
  MoveJ (Approach target)
  MoveL (Target 0)
  MoveL (Target 1)
  MoveL (Target 2)
  MoveL (Target 3)
  MoveL (Target 4)
  MoveL (Target 5)
  MoveL (Target 6)
  MoveL (Target 7)
  MoveL (Target 8)
  MoveL (Target 9)
  MoveL (Target 10)
  MoveL (Target 11)
  MoveL (Target 12)
  MoveL (Target 13)
  MoveL (Target 14)
  MoveL (Target 15)
  MoveL (Target 16)
  MoveL (Target 17)
  MoveL (Target 18)
  MoveL (Target 19)
  MoveL (Target 20)
  MoveL (Target 21)
  MoveL (Target 22)
  MoveL (Target 23)
  MoveL (Target 24)
  MoveL (Target 25)
  MoveL (Target 26)
  MoveL (Target 27)
  MoveL (Target 28)
  MoveL (Target 29)
  MoveL (Target 30)
  MoveL (Target 31)
  MoveL (Target 32)
  MoveL (Target 33)
  MoveL (Target 34)
  MoveL (Target 35)
  MoveL (Target 36)
  MoveL (Target 37)
  MoveL (Target 38)
  MoveL (Target 39)
  MoveL (Target 40)
  MoveL (Target 41)
  MoveL (Target 42)
  MoveL (Target 43)
  MoveL (Target 44)
  MoveL (Target 45)
  MoveL (Target 46)
  MoveL (Target 47)
  MoveL (Target 48)
  MoveL (Target 49)
  MoveL (Target 50)
  MoveL (Target 51)
  MoveL (Target 52)
  MoveL (Target 53)
  MoveL (Target 54)
  MoveL (Target 55)
  MoveL (Target 56)
  MoveL (Target 57)
  MoveL (Target 58)
  MoveL (Target 59)
  MoveL (Target 60)
  MoveL (Target 61)
  MoveL (Target 62)
  MoveL (Target 63)
  MoveL (Target 64)
  MoveL (Target 65)
  MoveL (Target 66)
  MoveL (Target 67)
  MoveL (Target 68)
  MoveL (Target 69)
  MoveL (Target 70)
  MoveL (Target 71)
  MoveL (Target 72)
  MoveL (Target 73)
  MoveL (Target 74)
  MoveL (Target 75)
  MoveL (Target 76)
  MoveL (Target 77)
  MoveL (Target 78)
  MoveL (Target 79)
  MoveL (Target 80)
  MoveL (Target 81)
  MoveL (Target 82)
  MoveL (Target 83)
  MoveL (Target 84)
  MoveL (Target 85)
  MoveL (Target 86)
  MoveL (Target 87)
  MoveL (Target 88)
  MoveL (Target 89)
  MoveL (Target 90)
  MoveL (Target 91)
  MoveL (Target 92)
  MoveL (Target 93)
  MoveL (Target 94)
  MoveL (Target 95)
  MoveL (Target 96)
  MoveL (Target 97)
  MoveL (Target 98)
  MoveL (Target 99)
  MoveL (Target 100)
  MoveL (Target 101)
  MoveL (Target 102)
  MoveL (Target 103)
  MoveL (Target 104)
  MoveL (Target 105)
  MoveL (Target 106)
  MoveL (Target 107)
  MoveL (Target 108)
  MoveL (Target 109)
  MoveL (Target 110)
  MoveL (Target 111)
  MoveL (Target 112)
  MoveL (Target 113)
  MoveL (Target 114)
  MoveL (Target 115)
  MoveL (Target 116)
  MoveL (Target 117)
  MoveL (Target 118)
  MoveL (Target 119)
  MoveL (Target 120)
  MoveL (Target 121)
  MoveL (Target 122)
  MoveL (Target 123)
  MoveL (Target 124)
  MoveL (Target 125)
  MoveL (Target 126)
  MoveL (Target 127)
  MoveL (Target 128)
  MoveL (Target 129)
  MoveL (Target 130)
  MoveL (Target 131)
  MoveL (Target 132)
  MoveL (Target 133)
  MoveL (Target 134)
  MoveL (Target 135)
  MoveL (Target 136)
  MoveL (Target 137)
  MoveL (Target 138)
  MoveL (Target 139)
  MoveL (Target 140)
  MoveL (Target 141)
  MoveL (Target 142)
  MoveL (Target 143)
  MoveL (Target 144)
  MoveL (Target 145)
  MoveL (Target 146)
  MoveL (Target 147)
  MoveL (Target 148)
  MoveL (Target 149)
  MoveL (Target 150)
  MoveL (Target 151)
  MoveL (Target 152)
  MoveL (Target 153)
  MoveL (Target 154)
  MoveL (Target 155)
  MoveL (Target 156)
  MoveL (Target 157)
  MoveL (Target 158)
  MoveL (Target 159)
  MoveL (Target 160)
  MoveL (Target 161)
  MoveL (Target 162)
  MoveL (Target 163)
  MoveL (Target 164)
